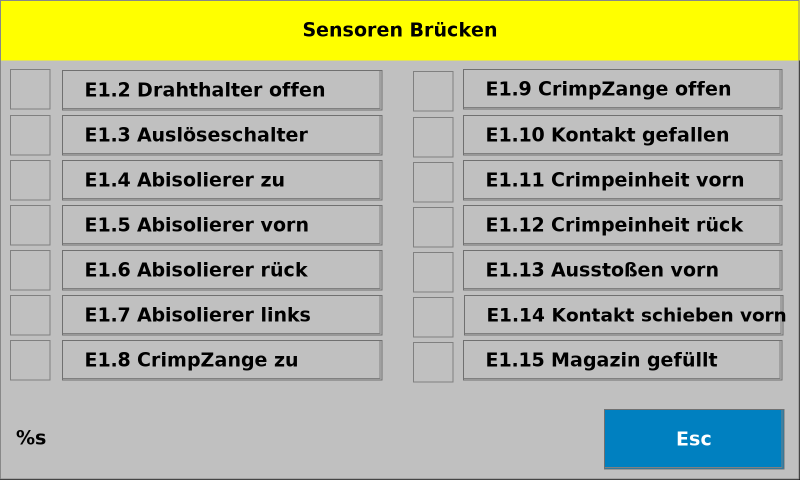
VISUALIZATION SensorBruecken  // 800x480
    Rectangle (0,0 800x480)
    Rectangle (0,0 800x60), "Sensoren Brücken"
    Button (604,409 180x60), "Esc"
        OnMouseUp: change screen: Previous Start
    Button (62,70 320x40), "E1.2 Drahthalter offen", tooltip "c", colour toggle: RVL.sBrDrahthalterIstOffen
        toggle RVL.sBrDrahthalterIstOffen
    Button (62,115 320x40), "E1.3 Auslöseschalter", colour toggle: RVL.sBrAusloeseSchalter
        toggle RVL.sBrAusloeseSchalter
    Button (62,160 320x40), "E1.4 Abisolierer zu", colour toggle: RVL.sBrAbisoliererIstZU
        toggle RVL.sBrAbisoliererIstZU
    Button (62,205 320x40), "E1.5 Abisolierer vorn", colour toggle: RVL.sBrAbisoliererIstVORN
        toggle RVL.sBrAbisoliererIstVORN
    Button (62,250 320x40), "E1.6 Abisolierer rück", colour toggle: RVL.sBrAbisoliererIstRUECK
        toggle RVL.sBrAbisoliererIstRUECK
    Button (62,295 320x40), "E1.7 Abisolierer links", colour toggle: RVL.sBrAbisoliererIstLINKS
        toggle RVL.sBrAbisoliererIstLINKS
    Button (62,340 320x40), "E1.8 CrimpZange zu", colour toggle: RVL.sBrCrimpZangeIstZU
        toggle RVL.sBrCrimpZangeIstZU
    Button (463,69 319x40), "E1.9 CrimpZange offen", colour toggle: RVL.sBrCrimpZangeIstOFFEN
        toggle RVL.sBrCrimpZangeIstOFFEN
    Button (463,115 319x40), "E1.10 Kontakt gefallen", colour toggle: RVL.sBrKontaktIstGefallen
        toggle RVL.sBrKontaktIstGefallen
    Button (463,160 319x40), "E1.11 Crimpeinheit vorn", colour toggle: RVL.sBrCrimpEinheitIstVORN
        toggle RVL.sBrCrimpEinheitIstVORN
    Button (464,295 319x40), "E1.14 Kontakt schieben vorn", colour toggle: RVL.sBrKontaktSchiebenVORN
        toggle RVL.sBrKontaktSchiebenVORN
    Button (463,250 319x40), "E1.13 Ausstoßen vorn", colour toggle: RVL.sBrAusstossenVORN
        toggle RVL.sBrAusstossenVORN
    Button (463,205 319x40), "E1.12 Crimpeinheit rück", colour toggle: RVL.sBrCrimpEinheitIstRUECK
        toggle RVL.sBrCrimpEinheitIstRUECK
    Button (463,340 319x40), "E1.15 Magazin gefüllt", colour toggle: RVL.sBrMagazinGEFUELLT
        toggle RVL.sBrMagazinGEFUELLT
    Rectangle (10,69 40x40), colour toggle: GVL.insecDrahthalterIstOffen
    Rectangle (10,115 40x40), colour toggle: GVL.insecAusloeseSchalter
    Rectangle (10,160 40x40), colour toggle: GVL.insecAbisoliererIstZU
    Rectangle (10,205 40x40), colour toggle: GVL.insecAbisoliererIstVORN
    Rectangle (10,250 40x40), colour toggle: GVL.insecAbisoliererIstRUECK
    Rectangle (10,295 40x40), colour toggle: GVL.insecAbisoliererIstLINKS
    Rectangle (10,340 40x40), colour toggle: GVL.insecCrimpZangeIstZU
    Rectangle (413,71 40x40), colour toggle: GVL.insecCrimpZangeIstOFFEN
    Rectangle (413,117 40x40), colour toggle: GVL.insecKontaktIstGefallen
    Rectangle (413,162 40x40), colour toggle: GVL.insecCrimpEinheitIstVORN
    Rectangle (413,207 40x40), colour toggle: GVL.insecCrimpEinheitIstRUECK
    Rectangle (413,252 40x40), colour toggle: GVL.insecAusstossenVORN
    Rectangle (413,297 40x40), colour toggle: GVL.insecKontaktSchiebenVORN
    Rectangle (413,342 40x40), colour toggle: GVL.insecMagazinGEFUELLT
    Rectangle (13,412 569x52), "%s", text list: 'BetrAnzeigeListe', text index: GVL.EinzelschrittIdx
END_VISUALIZATION

(* stored: Version 1.1.0.1, ProductVersion 3.1.4024.3
   Visu SensorBruecken: Id {2ef65297-a57b-476b-afac-b1860e6cfb23} *)
